Yaskawa INFORM job: BACK34IN.JBI

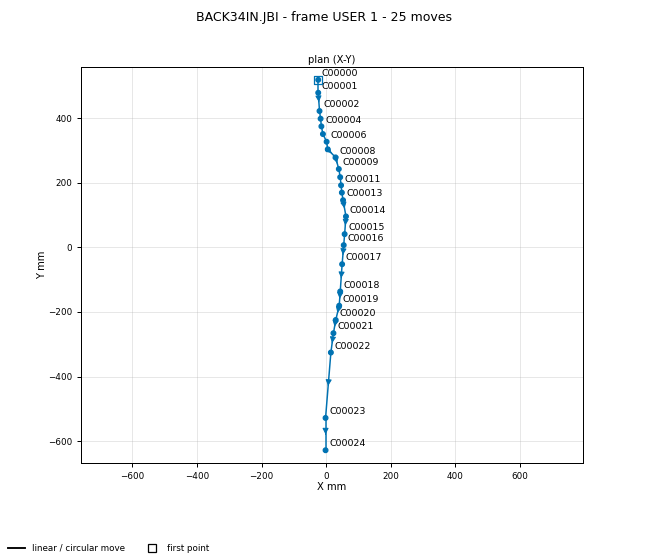
[picture p0: tool path of BACK34IN.JBI in frame USER 1, 25 of 25 moves have a stored position in this frame; points joined in program order, loops and branches not executed]
/JOB
//NAME BACK34IN
//POS
///NPOS 25,0,0,0,0,0
///TOOL 0
///USER 1
///POSTYPE USER
///RECTAN
///RCONF 1,0,0,0,0,0,0,0
C00000=-24.849,518.654,-65.000,180.00,-0.00,32.51
C00001=-24.849,478.654,-65.000,180.00,-0.00,32.51
C00002=-20.887,422.158,-65.000,180.00,-0.00,31.34
C00003=-17.524,398.421,-65.000,180.00,-0.00,30.58
C00004=-15.054,374.619,-65.000,180.00,-0.00,29.90
C00005=-10.311,350.877,-65.000,180.00,-0.00,28.81
C00006=1.114,327.102,-65.000,180.00,-0.00,26.47
C00007=4.618,303.585,-65.000,180.00,-0.00,25.44
C00008=28.749,278.624,-65.000,180.00,-0.00,20.11
C00009=38.873,242.564,-65.000,180.00,-0.00,17.07
C00010=43.195,217.342,-65.000,180.00,-0.00,15.42
C00011=45.871,192.223,-65.000,180.00,-0.00,14.04
C00012=48.304,169.480,-65.000,180.00,-0.00,12.63
C00013=52.055,146.025,-65.000,180.00,-0.00,10.48
C00014=61.042,95.787,-65.000,180.00,-0.00,3.26
C00015=56.875,41.056,-65.000,180.00,-0.00,2.91
C00016=54.092,6.921,-65.000,180.00,-0.00,2.94
C00017=49.123,-52.081,-65.000,180.00,-0.00,2.74
C00018=43.267,-136.511,-65.000,180.00,-0.00,3.17
C00019=40.106,-180.511,-65.000,180.00,-0.00,3.31
C00020=29.344,-224.793,-65.000,180.00,-0.00,1.46
C00021=22.249,-265.655,-65.000,180.00,-0.00,0.64
C00022=14.315,-325.472,-65.000,180.00,-0.00,0.09
C00023=-2.163,-528.009,-65.000,180.00,-0.00,0.09
C00024=-2.163,-628.009,-65.000,180.00,-0.00,0.09
//INST
///DATE 2020/12/14 17:40
///COMM Generated using RoboDK
///ATTR SC,RW,RJ
///GROUP1 RB1
NOP
'Using 0 (targets wrt base):
'0.0,0.0,0.0,0.0,0.0,0.0
'Tool 0 (0) should be close to
':
'0.0,0.0,0.0,0.0,0.0,0.0
'Program generated by RoboDK
MOVL C00000 V=150.0
MOVL C00001 V=178.0
MOVL C00002 V=178.0
MOVL C00003 V=178.0
MOVL C00004 V=178.0
MOVL C00005 V=178.0
MOVL C00006 V=178.0
MOVL C00007 V=178.0
MOVL C00008 V=178.0
MOVL C00009 V=178.0
MOVL C00010 V=178.0
MOVL C00011 V=178.0
MOVL C00012 V=178.0
MOVL C00013 V=178.0
MOVL C00014 V=178.0
MOVL C00015 V=178.0
MOVL C00016 V=178.0
MOVL C00017 V=178.0
MOVL C00018 V=178.0
MOVL C00019 V=178.0
MOVL C00020 V=178.0
MOVL C00021 V=178.0
MOVL C00022 V=178.0
MOVL C00023 V=178.0
MOVL C00024 V=178.0
END
